{attribute 'reflection'}
FUNCTION_BLOCK PUBLIC FB_DevBasicACAxis EXTENDS FB_DevBase
VAR_INPUT
	// ===== General Function input =====
		fCmdAcc			: LREAL := 15000;
		fCmdDecc		: LREAL := 15000; 
	// Manual control reference
		stManualCtrl	: UDT_ManualAxisCtrl ;
END_VAR
VAR_OUTPUT
	bHomed			: BOOL 	:= FALSE; 
	bMoving		: BOOL ; // Axis is moving
	bInPosition : BOOL ; // Axis is in position 
END_VAR
VAR
		AxisRef	: AXIS_REF ; // reference to AC axis
	// ===== HW Config Bits =====
		bIcfCmdVelocityRpm	: BOOL ; // input speeds in Rpm
		bIcfEnableForward 	: BOOL ; // Enable forward motion
 		bIcfEnablereverse	: BOOL ; // Enable reverse motion
		bIcfAlwaysEnable	: BOOL ; // 1 = Axis always enabled, 0 = Axis disabled at Idle 
		bIcfSimulationMode	: BOOL := FALSE ; // Simulation mode is active [default set to False] 
	// ===== Internal motion values ======
		fHomePosition		: LREAL := 0 ; // set position at homing
	// ====== Axis Settings ======
		fMaxVelo		: LREAL := 0 ; // Axis Maximum velocity
		fMaxAcc			: LREAL := 0 ; // Axis Maximum cceleration
		fMaxDec			: LREAL := 0 ; // axis Maxium deceleration 
		
		fSafeVeloLimit	: LREAL	:= 200; // Safe velocity limit 
		tEnableDelay	: TIME 	:= T#150MS	;
		tDisableDelay	: TIME 	:= T#500MS  ;
		
	// ====== Axis enable =====	
		bCmdEnableAxis 		: BOOL 	:= FALSE; // Command to enable the axis (External)
		bInternalEnable		: BOOL 	:= FALSE; // internal enable command (turns off after set time, and on at new motion command
		bDelayedEnable		: BOOL 	:= false; // Delayed enable signal for motion commands
		TonMotionEnable		: TON 			; // Timer on for motion command enable
		TofIntAxisEnable	: TOF  			; // Timer off for internal axis enable 
	// ===== Safe commands =====
		bCmdSafeStop	: BOOL ;
	// Motion commands 
		fbMcPower 			: MC_Power		;		// FB for enable and override
		fbMcReset 			: MC_Reset		;		// FB to reset axis
		fbSoeReset			: FB_SoEReset	; 		// FB to reset axis hardware
		fbMcHome			: MC_Home		;		// Fb to home Axis
		fbMcStop 			: MC_Stop		;		// FB to stop axis
		fbMcHalt			: MC_Halt		;		// FB to halt axis
		fbMcJog				: MC_Jog		;		// FB to Jog axis
		fbMcMoveVelocity	: MC_MoveVelocity;		// FB to move with specified velocity until Next command is given
	(* PtoP Motion move commands are in arrays so multiple commands can be stacked *) 
		fbMCMoveRelative	: ARRAY [0..1] OF MC_MoveRelative	;		// FB to move relative
		fbMcMoveAbsolute	: ARRAY [0..1] OF MC_MoveAbsolute	;		// FB to move axis (velocity movement)
		
	// Parameters 
		stMParMaxAcc : Udt_Parameter := (fMaximum := 999999, fMinimum := 0, fValue := 0)	; // Parameter for maximum acceleration
		stMParMaxDec : Udt_Parameter := (fMaximum := 999999, fMinimum := 0, fValue := 0)	; // Parameter for maximum Deceleration
		stMparMaxVelo: Udt_Parameter := (fMaximum := 999999, fMinimum := 0, fValue := 0)	; // Parameter for maximum velocity
		
	// Device feedback
		nActVelocity AT%I* : INT ; // actual speed of the motor
		nActPosition AT%I* : UDINT ; // Actual position of the motor

	// ===== Function execute triggers =====
		bExec_Reset			: BOOL := FALSE; // Execute reset
		bExec_Halt			: BOOL := FALSE; // Execute hold
		bExec_Home			: BOOL := FALSE; // Execute Home
		bExec_JogPositive	: BOOL := FALSE; // Execute Jog in positive direction
		bExec_JogNegative	: BOOL := FALSE; // Execute Jog in negative direction
		bExec_MoveVelocity	: BOOL := FALSE; // Execute move velocity
		arExec_MoveRelative	: ARRAY [0..1] OF BOOL ; // Execute move relative
		arExec_MoveAbs		: ARRAY [0..1] OF BOOL ; // Execute move absolute reverse
		

END_VAR

// Call base function
SUPER^(refFbFault := refFbFault);

// ==== Check if axis is initiated =====
IF NOT bInitOk THEN 
	RETURN ; 
END_IF

// ===== Execute safe functions =====
	ExecSafeFunctions(); 

// ==== Execute organizational functions =====
	ExecEnable();

// ==== execute motion functions =====
	CallMotionFunctions();

METHOD PRIVATE CallMotionFunctions : BOOL
VAR_INPUT
END_VAR
// ===== Check if safe to move =====
	IF bCmdSafeStop OR NOT bDelayedEnable THEN 
		RETURN ;
	END_IF

// ===== Homing functions =====
	ExecHome		(); 

// ===== Motion standstil commands =====
	ExecHalt		();

// ===== Motion move functions
	ExecJog			(); 
	ExecMoveAbsolute();
	ExecMoveRelative();
	ExecMoveVelocity();
END_METHOD

METHOD PUBLIC CmdHalt : BOOL
VAR_INPUT
	fDeceleration 	: LREAL := 0 ; // command deceleration
	mcBuffermode	: MC_BufferMode ; // Buffermode defines how the previous command is executed.
END_VAR
// Set command to true 
bExec_Halt 		:= TRUE ;
bInternalEnable	:= TRUE ;

// coppy parameters
fbMcHalt.Deceleration	:= fDeceleration;
fbMcHalt.BufferMode		:= mcBuffermode	;

// Set feedback output 
CmdHalt := fbMchalt.Active ;
END_METHOD

METHOD PUBLIC CmdHome : BOOL // start axis homing procedure
VAR_INPUT
	fPosition 		: LREAL := 0 ; // Homing position
	mcBufferMode	: MC_BufferMode := MC_BufferMode.MC_Aborting		; // Buffermode
END_VAR
// set command to true 
bExec_Home 		:= TRUE	; 
bInternalEnable	:= TRUE ;

// coppy parameters
fbMcHome.Position 	:= fPosition 	;
fbMcHome.BufferMode	:= mcBufferMode ;

// Set feedback output
CmdHome := fbMcHome.Done ;
END_METHOD

METHOD PUBLIC CmdJog : BOOL // Jog axis with variable speed. jog stops as soon as the command is false
VAR_INPUT
	fVelocity		: LREAL 	; // jog velocity can be adjusted as long as the command is active
	fPos			: LREAL 	; // Jog position or step size (if aplicable)
	bJogNegative 	: BOOL 		:= FALSE ; // jog in negative direction
	eJogmode		: E_JogMode := E_JogMode.MC_JOGMODE_CONTINOUS ; // jogmode [default MC_JOGMODE_CONTINOUS] 
END_VAR
// Velocity conversion from RPM to deg/sec
	IF bIcfCmdVelocityRpm THEN 
		fVelocity := Rpm_To_DegS(fVelocity);
	END_IF

// Set command to true
	IF fbMcJog.Velocity = fVelocity THEN // If command velocity changes, then set exec to false for one cycle to trigger new velocity so the jog follows the set velocity
		bExec_JogPositive	:= NOT bJogNegative ;
		bExec_JogNegative 	:= bJogNegative ;
	END_IF
	bInternalEnable			:= TRUE ;

// coppy parameters
	fbMcJog.Velocity	:= fVelocity 	;
	fbmcjog.Mode		:= eJogmode		;
	fbMcJog.Position	:= fPos			;

// Set feedback output 
	CmdJog := fbMcJog.Active ;
END_METHOD

METHOD PUBLIC CmdManual : BOOL
VAR
	eJogmode		: E_JogMode := E_JogMode.MC_JOGMODE_CONTINOUS ; // jogging mode 
END_VAR
// Enable axis for manual control
bCmdManual := TRUE ;

// set jog mode 
IF stManualCtrl.bCmdInching THEN 
	eJogmode := E_JogMode.MC_JOGMODE_INCHING ;
END_IF

// execute motion commands
IF stManualCtrl.bCmdJogForward OR stManualCtrl.bCmdJogReverse THEN 
	CmdJog (fVelocity := stManualCtrl.fVelocity, 
			fPos := stManualCtrl.fDistance, 
			bJogNegative := stManualCtrl.bCmdJogReverse, 
			eJogmode := eJogmode);
ELSIF stManualCtrl.bCmdToPos THEN 
	CmdMoveAbs( fPosition := stManualCtrl.fPosition, 
				fVelocity := stManualCtrl.fVelocity, 
				mcBuffermode := MC_BufferMode.MC_Aborting);
ELSIF stManualCtrl.bCmdHome THEN 
	CmdHome( fPosition := 0, mcBufferMode := MC_Aborting);
ELSE 
	CmdHalt( 	fDeceleration := fMaxDec * 0.9, 
				mcBuffermode := MC_BufferMode.MC_Aborting) ; 
END_IF
END_METHOD

METHOD PUBLIC CmdMoveAbs : BOOL // Move absolute command
VAR_INPUT
	fPosition	:	LREAL 	; // target position
	fVelocity	: 	LREAL 	; // Maximum velocity [units/sec]
	mcBuffermode: 	MC_BufferMode ; // Buffermode defines how the previous command is executed.
END_VAR
// Velocity conversion from RPM to deg/sec
	IF bIcfCmdVelocityRpm THEN 
		fVelocity := Rpm_To_DegS(fVelocity);
	END_IF

// Determine function for command stacking
	IF fbMcMoveAbsolute[0].Active THEN 
		arExec_MoveAbs[1] 				:= (fPosition <> fbMcMoveAbsolute[0].Position OR fVelocity <> fbMcMoveAbsolute[0].Velocity) ;
		fbMcMoveAbsolute[1].Position 	:= fPosition ;
		fbMcMoveAbsolute[1].Velocity 	:= fVelocity ; 
		fbMcMoveAbsolute[1].BufferMode 	:= mcBuffermode ;
	ELSE
		arExec_MoveAbs[0] 				:= (fPosition <> fbMcMoveAbsolute[1].Position OR fVelocity <> fbMcMoveAbsolute[1].Velocity) ;
		fbMcMoveAbsolute[0].Position 	:= fPosition ;
		fbMcMoveAbsolute[0].Velocity 	:= fVelocity ; 
		fbMcMoveAbsolute[0].BufferMode 	:= mcBuffermode ;
	END_IF

bInternalEnable	:= TRUE ;
// set feedback
IF arExec_MoveAbs[1] OR fbMcMoveAbsolute[1].Busy THEN 
	CmdMoveAbs :=	fbMcMoveAbsolute[1].Active ;
ELSE 
	CmdMoveAbs :=	fbMcMoveAbsolute[0].Active ;
END_IF
END_METHOD

METHOD CmdMoveRelative : BOOL // move relative command 
VAR_INPUT
	fDistance	:	LREAL 	; // target position
	fVelocity	: 	LREAL 	; // Maximum velocity [units/sec]
	mcBuffermode: 	MC_BufferMode ; // Buffermode defines how the previous command is executed.
END_VAR
// Velocity conversion from RPM to deg/sec
	IF bIcfCmdVelocityRpm THEN 
		fVelocity := Rpm_To_DegS(fVelocity);
	END_IF

// Determine function for command stacking
	IF fbMCMoveRelative[0].Active THEN 
		arExec_MoveRelative[1] := (fDistance <> fbMCMoveRelative[0].Distance OR fVelocity <> fbMCMoveRelative[0].Velocity) ;
		fbMCMoveRelative[1].Velocity	:= fVelocity 	;
		fbMCMoveRelative[1].Distance	:= fDistance	;
		fbMCMoveRelative[1].BufferMode	:= mcBuffermode	;
	ELSE 
		arExec_MoveRelative[0] := (fDistance <> fbMCMoveRelative[1].Distance OR fVelocity <> fbMCMoveRelative[1].Velocity) ;
		fbMCMoveRelative[0].Velocity	:= fVelocity 	;
		fbMCMoveRelative[0].Distance	:= fDistance	;
		fbMCMoveRelative[0].BufferMode	:= mcBuffermode	;
	END_IF

bInternalEnable	:= TRUE ;

// set feedback
IF arExec_MoveRelative[1] OR fbMCMoveRelative[1].Busy THEN 
	CmdMoveRelative :=	fbMCMoveRelative[1].Active ;
ELSE
	CmdMoveRelative :=	fbMCMoveRelative[0].Active ;
END_IF
END_METHOD

METHOD PUBLIC CmdMoveVelocity : BOOL // Move with set velocity until stopped
VAR_INPUT
	fVelocity	: 	LREAL 	; // Maximum velocity [units/sec]
	mcDirection : 	MC_Direction := MC_Direction.MC_Positive_Direction ; // Direction of movement mc_direction [ deafult mc_positive_direction]
	mcBuffermode: 	MC_BufferMode ; // Buffermode defines how the previous command is executed.
END_VAR
// Velocity conversion from RPM to deg/sec
	IF bIcfCmdVelocityRpm THEN 
		fVelocity := Rpm_To_DegS(fVelocity);
	END_IF

// Set command to true 
	bExec_MoveVelocity 	:= TRUE ;
	bInternalEnable		:= TRUE ;

// coppy parameters
	fbMcMoveVelocity.Velocity	:= fVelocity 	;
	fbMcMoveVelocity.Direction 	:= mcDirection	;
	fbMcMoveVelocity.BufferMode	:= mcBuffermode	;

// Set feedback output 
	CmdMoveVelocity := fbMcMoveVelocity.Active ;
END_METHOD

METHOD PUBLIC CmdReset : BOOL
VAR_INPUT
END_VAR
// Set reset axis to true 				
	bExec_Reset 	:= TRUE ; 
	bInternalEnable	:= TRUE ;
	
// Set feedback output 
	CmdReset := fbMcReset.Done ;
END_METHOD

METHOD PUBLIC CmdSafeStop : BOOL
VAR_INPUT
END_VAR
// Set safestop command
bCmdSafeStop := TRUE ; 

// Set feedback output 
CmdSafeStop := bIsSafe OR NOT bInitOk;
END_METHOD

METHOD PRIVATE ExecEnable : BOOL
VAR_INPUT
END_VAR
// ===== Set axis enable ======
IF NOT bEnable AND NOT bCmdManual AND nActVelocity <> 0 THEN
	CmdHalt(fDeceleration := fCmdDecc, mcBuffermode := MC_BufferMode.MC_Aborting);
ELSE 
	bCmdEnableAxis	:= bEnable OR bCmdManual ;
	bCmdManual := FALSE ;
END_IF

// ===== Check if axis is bussy with a command =====
	bInternalEnable	S= bIcfAlwaysEnable ; // always enable axis if configured
	
// ===== Axis disable timer after last command =====
	TofIntAxisEnable (	IN:= bInternalEnable, PT := tDisableDelay);

// ===== Enable drive =====
	fbMcPower(	Axis			:= AxisRef , 
				Enable			:= bCmdEnableAxis AND TofIntAxisEnable.Q, 
				Enable_Positive	:= bIcfEnableForward, 
				Enable_Negative	:= bIcfEnablereverse, 
				Override		:= 100 );  
				
// ===== Reset internal enable signal =====
	bInternalEnable := FALSE ; 	

// ===== Delayed enable function =====	
	TonMotionEnable(IN := fbMcPower.Active, PT := tEnableDelay);
	bDelayedEnable := TonMotionEnable.Q ;	


IF fbMcPower.Error THEN 
	bErrorActive			:= TRUE							;
	stFault.Active 			:= TRUE 						;
	stFault.MessageNumber	:= E_MessageNumbers.FF_AxisFault;
	stFault.Discription		:= CONCAT('Enable Fault ', UDINT_TO_STRING(fbMcPower.ErrorID));				;
	stFault.FaultType		:= E_FaultTypes.FF				;
END_IF
END_METHOD

METHOD PRIVATE ExecHalt : BOOL
VAR_INPUT
END_VAR
// ==== Execute halt function ===== 
fbMcHalt (	Axis 		:= AxisRef,
			Execute 	:= bExec_Halt );

// ===== reset command =====
	bExec_Halt := FALSE ;
	bInternalEnable := fbMcHalt.Busy ;			
	
// Halt fault handling 
	IF fbMcHalt.Error THEN 
		bErrorActive			:= TRUE							;
		stFault.Active 			:= TRUE 						;
		stFault.MessageNumber	:= E_MessageNumbers.FF_AxisFault;
		stFault.Discription		:= CONCAT('Halt Fault ', UDINT_TO_STRING(fbMcHalt.ErrorID));				;
		stFault.FaultType		:= E_FaultTypes.FF				;
	END_IF
END_METHOD

METHOD PRIVATE ExecHome : BOOL
VAR_INPUT
END_VAR
// ==== execute homing function =====
	fbMcHome(	Axis			:= AxisRef,
				Execute			:= bExec_Home,
				HomingMode		:= MC_DefaultHoming ); 
			
// Reset exec command 
	bExec_Home 	:= FALSE ;
	bHomed		S= fbMcHome.Done ;	
	bInternalEnable := fbMcHome.Busy ;			
				
// fault handling 
	IF fbMcHome.Error THEN 
		bErrorActive			:= TRUE							;
		stFault.Active 			:= TRUE 						;
		stFault.MessageNumber	:= E_MessageNumbers.FF_AxisFault;
		stFault.Discription		:= CONCAT('Homing Fault ', UDINT_TO_STRING(fbMcHome.ErrorID));				;
		stFault.FaultType		:= E_FaultTypes.FF				;
	END_IF
END_METHOD

METHOD PRIVATE ExecJog : BOOL
VAR_INPUT
END_VAR
// ===== Execute Jog function =====
	// function call
	fbMcJog (	Axis 		:= AxisRef,
				JogForward	:= bExec_JogPositive,
				JogBackwards:= bExec_JogNegative,
				Acceleration:= fCmdAcc,
				Deceleration:= fCmdDecc );

// ===== reset command =====
	bExec_JogPositive 	:= FALSE  ;
	bExec_JogNegative	:= FALSE  ;
	bInternalEnable		:= fbMcJog.Busy; 

// Jog fault handling 
	IF fbMcJog.Error THEN 
		bErrorActive			:= TRUE							;
		stFault.Active 			:= TRUE 						;
		stFault.MessageNumber	:= E_MessageNumbers.FF_AxisFault;
		stFault.Discription		:= CONCAT('Jog Fault ', UDINT_TO_STRING(fbMcJog.ErrorID));				;
		stFault.FaultType		:= E_FaultTypes.FF				;
	END_IF
END_METHOD

METHOD PRIVATE ExecMoveAbsolute : BOOL
VAR_INPUT
END_VAR
VAR
	i : UDINT := 0 ;
END_VAR
// ==== execute move absolute function =====
FOR i := 0 TO 1 DO 
	// function call
	fbMcMoveAbsolute[i](	Axis 		:= AxisRef,
							Execute 	:= arExec_MoveAbs[i],
							Acceleration:= fCmdAcc,
							Deceleration:= fCmdDecc );  
	// reset Exec command 
	arExec_MoveAbs[i] := FALSE ; 
	bInternalEnable := fbMcMoveAbsolute[i].Busy ;			

	// If function is done then reset command values
	IF fbMcMoveAbsolute[i].Done THEN 
		fbMcMoveAbsolute[i].Velocity	:= 0 ;
		fbMcMoveAbsolute[i].Position	:= 0 ; 
	END_IF
	
	// fault handling 
	IF fbMcMoveAbsolute[i].Error THEN 
		bErrorActive			:= TRUE							;
		stFault.Active 			:= TRUE 						;
		stFault.MessageNumber	:= E_MessageNumbers.FF_AxisFault;
		stFault.Discription		:= CONCAT('Move absolute Fault ', UDINT_TO_STRING(fbMcMoveAbsolute[i].ErrorID));				;
		stFault.FaultType		:= E_FaultTypes.FF				;
	END_IF
END_FOR
END_METHOD

METHOD PRIVATE ExecMoveRelative : BOOL
VAR_INPUT
END_VAR
VAR
	i : UDINT := 0 ;
END_VAR
// ===== Execute move relative function ======
FOR i := 0 TO 1 DO 
	// function call
	fbMCMoveRelative[i](	Axis 		:= AxisRef,
							Execute		:= arExec_MoveRelative[i],
							Acceleration:= fCmdAcc,
							Deceleration:= fCmdDecc );
	// reset Exec command 
	arExec_MoveRelative[i] := FALSE ; 
	bInternalEnable := fbMCMoveRelative[i].Busy ;			

	// If function is done then reset command values
	IF fbMCMoveRelative[i].Done THEN 
		fbMCMoveRelative[i].Velocity	:= 0 ;
		fbMCMoveRelative[i].Distance	:= 0 ; 
	END_IF
	
	// fault handling 
	IF fbMCMoveRelative[i].Error THEN 
		bErrorActive			:= TRUE							;
		stFault.Active 			:= TRUE 						;
		stFault.MessageNumber	:= E_MessageNumbers.FF_AxisFault;
		stFault.Discription		:= CONCAT('Move relative Fault ', UDINT_TO_STRING(fbMCMoveRelative[i].ErrorID));				;
		stFault.FaultType		:= E_FaultTypes.FF			;
	END_IF
END_FOR
END_METHOD

METHOD PRIVATE ExecMoveVelocity : BOOL
VAR_INPUT
END_VAR
// ===== Execute move velocity function =====
// function call
fbMcMoveVelocity (	Axis 		:= AxisRef,
					Execute		:= bExec_MoveVelocity,
					Acceleration:= fCmdAcc,
					Deceleration:= fCmdDecc );

// ===== reset command =====
bExec_MoveVelocity := FALSE ;
bInternalEnable		:= fbMcMoveVelocity.Busy;
	
// Halt fault handling 
IF fbMcHalt.Error THEN 
	bErrorActive			:= TRUE							;
	stFault.Active 			:= TRUE 						;
	stFault.MessageNumber	:= E_MessageNumbers.FF_AxisFault;
	stFault.Discription		:= CONCAT('Move velocity Fault ', UDINT_TO_STRING(fbMcMoveVelocity.ErrorID));				;
	stFault.FaultType		:= E_FaultTypes.FF				;
END_IF
END_METHOD

METHOD PRIVATE ExecReset : BOOL
VAR_INPUT
END_VAR
IF  nActVelocity <> 0 AND bExec_Reset THEN // If the axis is still moving execute safe stop first
	CmdSafeStop();
	RETURN;
END_IF

// perform reset 
	fbMcReset	( 	Execute	:= bexec_reset AND NOT fbSoeReset.Busy,
					Axis	:= AxisRef ); 
					
// ===== reset command =====
	bExec_Reset := FALSE ;
	
// ===== reset internal fault bits and stop bits =====
	bErrorActive 			:= FALSE ; 
	
// ===== reset safe commands ======
	bCmdSafeStop	:= FALSE ; 
	
// Reset fault handling 
	IF fbSoeReset.Error OR fbMcReset.Error THEN 
		bErrorActive			:= TRUE							;
		stFault.Active 			:= TRUE 						;
		stFault.MessageNumber	:= E_MessageNumbers.FF_AxisFault;
		stFault.Discription		:= CONCAT('Reset Fault ', UDINT_TO_STRING(fbMcReset.ErrorID))			;
		stFault.FaultType		:= E_FaultTypes.FF				;
	END_IF
END_METHOD

METHOD PRIVATE ExecSafeFunctions : BOOL
VAR_INPUT
END_VAR
// ==== Stop when safety is not ok =====
	bCmdSafeStop := NOT bSafetyOk ;

// ==== Safe operation functions (overrule all other motion functions) =====
	fbMcStop( 	Axis 			:= AxisRef		,
				Execute 		:= bCmdSafeStop	,
				Deceleration	:= fMaxDec		);
	
	// Reset axis command			
	bCmdSafeStop 	R= fbMcStop.Done ;
	
// Safestop fault handling 
	IF fbMcStop.Error THEN 
		bErrorActive			:= TRUE							;
		stFault.Active 			:= TRUE 						;
		stFault.MessageNumber	:= E_MessageNumbers.FF_AxisFault;
		stFault.Discription		:= CONCAT('Safe stop axis fault ', UDINT_TO_STRING(fbMcStop.ErrorID));				;
		stFault.FaultType		:= E_FaultTypes.FF				;
	END_IF

// ===== Dev is safe feedback =====
bIsSafe := NOT bCmdEnableAxis  ;
END_METHOD

METHOD PUBLIC Init : BOOL
VAR_INPUT
	// Message location data
	nId			: UDINT ; // Identification number of object
	nParentId	: UDINT ; // Id of higher level If aplicable (0 = no parent)
	// Config Bits
	bIcfCmdVelocityRpm	: BOOL := FALSE ; // input speeds in Rpm
	bIcfEnableForward 	: BOOL := TRUE 	; // Enable forward motion
	bIcfEnablereverse	: BOOL := TRUE 	; // Enable reverse motion
	bIcfAlwaysEnable	: BOOL := FALSE ; // 1 = Axis always enabled, 0 = Axis disabled at Idle 
	bIcfSimulationMode	: BOOL := FALSE ; // Simulation mode is active [default set to False] Used for testing without hardware present 
	
	fHomePosition		: LREAL := 0 	; // set position at homing
	fSafeVeloLimit		: LREAL	:= 360 	; // safe velocity limit [deg/sec]
	nEncTurnoverVal 	: LREAL := 360	; // encoder turnover value 
	tEnableDelay		: time 	:= T#0MS; // Time between axis enable command and motion command execution (0 := no delay active)	
	tDisabledelay		: TIME 	:= T#100MS; // Axis idle time before axis is disabled 
END_VAR
VAR 
	bActParamValid 		: BOOL ; // Parameter read is valid 
END_VAR
// Calculate device number
	ExecIdentifyDevice(nId,nParentId,E_ComponentTypes.Axis);

// ===== Message data set =====
	stFault.ComponentType		:= E_ComponentTypes.Axis ;
	
// ===== Write parameters =====
	stMParMaxAcc.nNumber		:= nLocationId + 1;
	stMParMaxAcc.sDiscription 	:= CONCAT(STR1 := sName, STR2:= ' hardware maximum accaleration (0 = HWMaximum)'); 
	stMParMaxAcc.sName			:= CONCAT(STR1 := sName, STR2:= 'Hard max aceleration');
	stMParMaxAcc.sType			:= 'MPar';
	stMParMaxAcc.sUnit			:= 'Units/Sec^2';
	
	stMParMaxDec.nNumber		:= nLocationId + 2;
	stMParMaxDec.sDiscription 	:= CONCAT(STR1 := sName, STR2:= ' hardware maximum deceleration(0 = HWMaximum)'); 
	stMParMaxDec.sName			:= CONCAT(STR1 := sName, STR2:= 'Hard max deceleration');
	stMParMaxDec.sType			:= 'MPar';
	stMParMaxDec.sUnit			:= 'Units/Sec^2';
	
	stMparMaxVelo.nNumber		:= nLocationId + 3;
	stMparMaxVelo.sDiscription 	:= CONCAT(STR1 := sName, STR2:= ' hardware maximum velocity'); 
	stMparMaxVelo.sName			:= CONCAT(STR1 := sName, STR2:= 'Hard max velocity');
	stMparMaxVelo.sType			:= 'MPar';
	stMparMaxVelo.sUnit			:= 'Units/Sec';

	refFbParHandler.CmdAddParameter(refParameter := stMParMaxAcc);
	refFbParHandler.CmdAddParameter(refParameter := stMParMaxDec);
	refFbParHandler.CmdAddParameter(refParameter := stMparMaxVelo);

// ===== set axis configuration =====	
	fMaxAcc	:= stMParMaxAcc.fValue;
	fMaxDec	:= stMParMaxDec.fValue;	
	fMaxVelo:= stMparMaxVelo.fValue;

	fCmdAcc 		:= fMaxAcc;
	fCmdDecc		:= fMaxDec;
// ===== Configure Axis =====
	// ***** Config Bits *****
		THIS^.bIcfCmdVelocityRpm	:= bIcfCmdVelocityRpm	; // Enable speed inputs in Rpm
		THIS^.bIcfEnableForward 	:= bIcfEnableForward 	; // Enable forward motion
		THIS^.bIcfEnablereverse		:= bIcfEnablereverse	; // Enable reverse motion
		THIS^.bIcfAlwaysEnable		:= bIcfAlwaysEnable		; // Always enable motor and brake if safety is ok
		THIS^.bIcfSimulationMode	:= bIcfSimulationMode 	; // Simulation mode is active [default set to False] 

	// ***** config homing Mode ***** 
 		THIS^.fHomePosition			:= fHomePosition;
	// ***** Velocity settings *****
		THIS^.fSafeVeloLimit 		:= fSafeVeloLimit ; // set maximum safe velocity	
	// ***** Time delay enable off *****
		THIS^.tEnableDelay		:= tEnableDelay	;
		THIS^.tDisableDelay 	:= tDisabledelay ;		

// ===== Set device type for manual control =====
	eDevType := E_Devices.Axis ;
		
// ===== reset axis state indicators ======
	bErrorActive 	:= FALSE;

// ====== Set init to done =======
	bInitOk	:= TRUE ;
END_METHOD

END_FUNCTION_BLOCK

(* stored: Version 1.1.0.1, ProductVersion 3.1.4024.5
   POU FB_DevBasicACAxis: Id {399212fc-3ad5-0237-1986-954c33e143fb}, SpecialFunc None
   Folder Commands: Id {e09297dc-c0aa-084c-2068-146d286afe03}
   Folder Private: Id {eedcaa3e-644e-09d2-2c97-9667d8fb0b6d}
   Folder Motion: Id {c83b6963-b999-0671-1f0a-c1203bae4a7b}
   Method CallMotionFunctions: Id {df6778e1-9f18-0c6d-097d-55e6d2427ff8}
   Method CmdHalt: Id {5fb82a80-5ffd-4f72-a47d-3a79f4d895b6}
   Method CmdHome: Id {3e65844c-78e5-091f-07c7-94c1b81b1a5a}
   Method CmdJog: Id {98cb74ae-0596-0a13-381d-d275b1843d1b}
   Method CmdManual: Id {3ce40203-b4d2-0a5e-34ee-d827b0a8f117}
   Method CmdMoveAbs: Id {c8a2c223-ab9e-00a2-1b56-623ff0fdbb39}
   Method CmdMoveRelative: Id {1795bbb4-c9d8-0ad1-361b-9df2709687fb}
   Method CmdMoveVelocity: Id {da29b8c2-802c-0e9d-24ac-ab6110610414}
   Method CmdReset: Id {ba035b82-611e-08e7-27b1-b4a38a3b499d}
   Method CmdSafeStop: Id {1272661a-b4ca-456b-a28d-d7b759e2f06a}
   Method ExecEnable: Id {090a0249-1749-0de7-24c6-e8a259604e68}
   Method ExecHalt: Id {1dacf53f-a12f-0750-236b-ec8fbb2b7997}
   Method ExecHome: Id {b92b1e44-987c-021c-13a3-ad0cde1da971}
   Method ExecJog: Id {29ca9d00-0145-0213-0626-7b8b0955b474}
   Method ExecMoveAbsolute: Id {cbfacbc8-a3df-0e23-027d-0daf2a93e334}
   Method ExecMoveRelative: Id {dd527bc6-4687-0467-3966-04400a33b2aa}
   Method ExecMoveVelocity: Id {00275b2c-af05-0c37-1b38-b1989240cb13}
   Method ExecReset: Id {2fec5393-4f47-011f-1ff8-817d4f397ca7}
   Method ExecSafeFunctions: Id {73a129ec-3a9f-0fc1-0be4-220de2bfc911}
   Method Init: Id {d9ee605e-1b43-0849-35b2-d86a67775109} *)
